(*
 *****************************************************************************
 * timeGetDcTime: Get TwinCAT DC time from UTC time
 *
 *  IN   vltUTC: UTC time 
 *  OUT  dcTIME: TwinCAT DC time
 ***************************************************************************** 
 *)
FUNCTION F_timeGetDcTime : ULINT
VAR_INPUT
	ut:	T_TIMEVAL;
END_VAR
VAR
	val:   	ULINT := 0;
END_VAR

(*
HRESULT timeGetDcTime(vltTIMEVAL vltUTC, LONGLONG *dcTime)
{
	HRESULT hr = S_OK; 
	LONGLONG val = 0;
	val = vltUTC.tv_sec * 1000000000;
	val -= OFFSET_UNIX;
	*dcTime = val + vltUTC.tv_usec * 1000;
	return hr;
}
*)
val	:= ut.tv_sec * 1000000000;
val := val - DINT_TO_ULINT(GCL.C_OFFSET_UNIX);

F_timeGetDcTime	:= val + DINT_TO_ULINT(ut.tv_usec) * 1000;

END_FUNCTION

(* stored: Version 1.1.0.1, ProductVersion 3.1.4022.9
   POU F_timeGetDcTime: Id {7186f94b-4e7e-43fa-be53-91561abe491a}, SpecialFunc None *)
